FUNCTION_BLOCK Q_ListItem (* Command change list item ( Part 6 - F.42 ) *)
  (* Standard: ISO 11783-6; Description: This command is used to change a list item in a list input object. Return values iso_s16 - E_NO_ERR - OK - E_OVERFLOW - buffer overflow - E_NOACT - Command not possible in current state - E_NO_INSTANCE - No VT client available *)
  (* Version 1.0, 2022-07-08, franz *)
  (* Documentation:
  This command is used to change a list item in a list input object.
   Return values
   iso_s16
    - E_NO_ERR - OK
   - E_OVERFLOW - buffer overflow
   - E_NOACT - Command not possible in current state
   - E_NO_INSTANCE - No VT client available
  *)
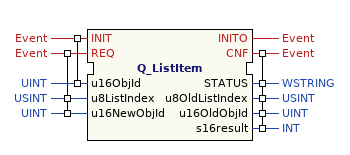
  EVENT_INPUT
    INIT WITH u16ObjId; (* Service Initialization *)
    REQ WITH u8ListIndex, u16NewObjId; (* Service Request *)
  END_EVENT
  EVENT_OUTPUT
    INITO; (* Initialization Confirm *)
    CNF WITH STATUS, s16result, u8OldListIndex, u16OldObjId; (* Confirmation of Requested Service *)
  END_EVENT
  VAR_INPUT
    u16ObjId : UINT; (* Object ID *)
    u8ListIndex : USINT; (* List index (-&gt; see list) *)
    u16NewObjId : UINT; (* New object ID or 0xFFFF to set empty *)
  END_VAR
  VAR_OUTPUT
    STATUS : WSTRING; (* Service Status *)
    u8OldListIndex : USINT; (* Old list index (-&gt; see list) *)
    u16OldObjId : UINT; (* Old object ID or 0xFFFF to set empty *)
    s16result : INT; (* retval see description *)
  END_VAR
END_FUNCTION_BLOCK
